// TwinCAT 3 PLC project PLC1
// Title: XPlanar Example Project
// Company: Beckhoff Automation LLC
// ProjectVersion: 1.0.0
// ProgramVersion: 3.1.4023.0
// libraries:
//   SPT Base Types, * (Beckhoff Automation LLC)
//   SPT Event Logger, * (Beckhoff Automation LLC)
//   SPT_XPlanar, * (Beckhoff Automation LLC)
//   Tc2_EtherCAT, * (Beckhoff Automation GmbH)
//   Tc2_Math, * (Beckhoff Automation GmbH)
//   Tc2_Standard, * (Beckhoff Automation GmbH)
//   Tc2_System, * (Beckhoff Automation GmbH)
//   Tc3_EventLogger, * (Beckhoff Automation GmbH)
//   Tc3_Module, * (Beckhoff Automation GmbH)
//   Tc3_PackML_V2, * (Beckhoff Automation GmbH)
//   Tc3_XPlanarUtility, * (Beckhoff Automation GmbH & Co. KG)
//   Tc3_Mc3PlanarMotion,newest,Beckhoff Automation GmbH
//   Tc3_Physics,newest,Beckhoff Automation GmbH
//   Tc3_XPlanarStandard,newest,Beckhoff Automation GmbH
//   VisuSymbols,3.5.10.0,System
// project tree:
//   / GlobalTextList.TcGTLO, MAIN.TcPOU, NextMinorStep.TcPOU, NextStep.TcPOU, PlcTask.TcTTO, StationList_TextList.TcTLO, Visualization Manager.TcVMO (not stored)
//   Machine/EquipmentModules/CustomStations/ FB_DecisionStation.TcPOU, FB_SpinStation.TcPOU
//   Machine/EquipmentModules/ FB_XPlanar_EM.TcPOU
//   Machine/ FB_Machine.TcPOU
//   Machine/VISUs/VisuOjects/ V_MachineModule.TcVIS, V_Module.TcVIS, V_Mover.TcVIS, V_RotaryAxis.TcVIS, V_Station.TcVIS
//   Machine/VISUs/ V_Main.TcVIS
// real-time tasks:
//   TASK PlcTask: cycle T#10ms, priority 20, ADS port 350
//   TASK Job Task: cycle default, priority 15
//   TASK MC-Task (MET): cycle T#2ms, priority 13, ADS port 521
//   TASK MC-Task (MPT): cycle T#10ms, priority 14, ADS port 531
//   TASK XPlanar Task11: cycle T#500us, priority 2, ADS port 352
//   TASK XPlanar Task6: cycle T#250us, priority 1, ADS port 351
//   TASK XPlanar Task7: cycle T#250us, priority 12, ADS port 353
//   TASK XPlanar Task3: cycle T#250us, priority 5, ADS port 354
//   TASK XPlanar Task4: cycle T#250us, priority 9, ADS port 355
//   TASK XPlanar Task5: cycle T#250us, priority 10, ADS port 356
// variable links:
//   XPlanar MC Project/Axes/Mover4220_1 <-> TcCOM Objects/XPlanar/Mover4220_1
//     McToIo/STD <-> InputsFromNC3/NC3ToHW
//   XPlanar MC Project/Axes/Mover4220_2 <-> TcCOM Objects/XPlanar/Mover4220_2
//     IoToMc/STD <-> OutputsToNC3/HWToNC3
//   XPlanar MC Project/Axes/Mover4220_3 <-> TcCOM Objects/XPlanar/Mover4220_3
//     IoToMc/STD <-> OutputsToNC3/HWToNC3
//   XPlanar MC Project/Axes/Mover4220_4 <-> TcCOM Objects/XPlanar/Mover4220_4
//     IoToMc/STD <-> OutputsToNC3/HWToNC3
//   PLC1/PLC1 Instance <-> XPlanar MC Project/Axes/Mover4220_1
//     PlcTask Inputs/MAIN.Machine.XPlanar.Movers[1]._Mover.stMoverRef.MCTOPLC/ACT <-> McToPlc/ACT
//     PlcTask Inputs/MAIN.Machine.XPlanar.Movers[1]._Mover.stMoverRef.MCTOPLC/COORDMODE <-> McToPlc/COORDMODE
//     PlcTask Inputs/MAIN.Machine.XPlanar.Movers[1]._Mover.stMoverRef.MCTOPLC/SET <-> McToPlc/SET
//     PlcTask Inputs/MAIN.Machine.XPlanar.Movers[1]._Mover.stMoverRef.MCTOPLC/SETONTRACK <-> McToPlc/SETONTRACK
//     PlcTask Inputs/MAIN.Machine.XPlanar.Movers[1]._Mover.stMoverRef.MCTOPLC/STD <-> McToPlc/STD
//     PlcTask Outputs/MAIN.Machine.XPlanar.Movers[1]._Mover.stMoverRef.PLCTOMC/STD <-> PlcToMc/STD
//   PLC1/PLC1 Instance <-> XPlanar MC Project/Axes/Mover4220_2
//     PlcTask Inputs/MAIN.Machine.XPlanar.Movers[2]._Mover.stMoverRef.MCTOPLC/ACT <-> McToPlc/ACT
//     PlcTask Inputs/MAIN.Machine.XPlanar.Movers[2]._Mover.stMoverRef.MCTOPLC/COORDMODE <-> McToPlc/COORDMODE
//     PlcTask Inputs/MAIN.Machine.XPlanar.Movers[2]._Mover.stMoverRef.MCTOPLC/SET <-> McToPlc/SET
//     PlcTask Inputs/MAIN.Machine.XPlanar.Movers[2]._Mover.stMoverRef.MCTOPLC/SETONTRACK <-> McToPlc/SETONTRACK
//     PlcTask Inputs/MAIN.Machine.XPlanar.Movers[2]._Mover.stMoverRef.MCTOPLC/STD <-> McToPlc/STD
//     PlcTask Outputs/MAIN.Machine.XPlanar.Movers[2]._Mover.stMoverRef.PLCTOMC/STD <-> PlcToMc/STD
//   PLC1/PLC1 Instance <-> XPlanar MC Project/Axes/Mover4220_3
//     PlcTask Inputs/MAIN.Machine.XPlanar.Movers[3]._Mover.stMoverRef.MCTOPLC/ACT <-> McToPlc/ACT
//     PlcTask Inputs/MAIN.Machine.XPlanar.Movers[3]._Mover.stMoverRef.MCTOPLC/COORDMODE <-> McToPlc/COORDMODE
//     PlcTask Inputs/MAIN.Machine.XPlanar.Movers[3]._Mover.stMoverRef.MCTOPLC/SET <-> McToPlc/SET
//     PlcTask Inputs/MAIN.Machine.XPlanar.Movers[3]._Mover.stMoverRef.MCTOPLC/SETONTRACK <-> McToPlc/SETONTRACK
//     PlcTask Inputs/MAIN.Machine.XPlanar.Movers[3]._Mover.stMoverRef.MCTOPLC/STD <-> McToPlc/STD
//     PlcTask Outputs/MAIN.Machine.XPlanar.Movers[3]._Mover.stMoverRef.PLCTOMC/STD <-> PlcToMc/STD
//   PLC1/PLC1 Instance <-> XPlanar MC Project/Axes/Mover4220_4
//     PlcTask Inputs/MAIN.Machine.XPlanar.Movers[4]._Mover.stMoverRef.MCTOPLC/ACT <-> McToPlc/ACT
//     PlcTask Inputs/MAIN.Machine.XPlanar.Movers[4]._Mover.stMoverRef.MCTOPLC/COORDMODE <-> McToPlc/COORDMODE
//     PlcTask Inputs/MAIN.Machine.XPlanar.Movers[4]._Mover.stMoverRef.MCTOPLC/SET <-> McToPlc/SET
//     PlcTask Inputs/MAIN.Machine.XPlanar.Movers[4]._Mover.stMoverRef.MCTOPLC/SETONTRACK <-> McToPlc/SETONTRACK
//     PlcTask Inputs/MAIN.Machine.XPlanar.Movers[4]._Mover.stMoverRef.MCTOPLC/STD <-> McToPlc/STD
//     PlcTask Outputs/MAIN.Machine.XPlanar.Movers[4]._Mover.stMoverRef.PLCTOMC/STD <-> PlcToMc/STD
//   PLC1/PLC1 Instance <-> XPlanar MC Project/Groups/Environment
//     PlcTask Inputs/MAIN.Machine.XPlanar.XPlanarTable.XPlanarSystem.environment.MCTOPLC_STD <-> McToPlc/STD
//   PLC1/PLC1 Instance <-> XPlanar MC Project/Groups/Group3 (Planar Track)
//     PlcTask Inputs/MAIN.Machine.XPlanar.Tracks[1].TrackStandard.stTrackRef.MCTOPLC_STD <-> McToPlc/STD
//   PLC1/PLC1 Instance <-> XPlanar MC Project/Groups/Group4 (Planar Track)
//     PlcTask Inputs/MAIN.Machine.XPlanar.Tracks[2].TrackStandard.stTrackRef.MCTOPLC_STD <-> McToPlc/STD
//   PLC1/PLC1 Instance <-> XPlanar MC Project/Groups/Group5 (Planar Track)
//     PlcTask Inputs/MAIN.Machine.XPlanar.Tracks[3].TrackStandard.stTrackRef.MCTOPLC_STD <-> McToPlc/STD
//   PLC1/PLC1 Instance <-> XPlanar MC Project/Groups/Group6 (Planar Track)
//     PlcTask Inputs/MAIN.Machine.XPlanar.Tracks[4].TrackStandard.stTrackRef.MCTOPLC_STD <-> McToPlc/STD
//   PLC1/PLC1 Instance <-> XPlanar MC Project/Groups/XPlanar
//     PlcTask Inputs/MAIN.Machine.XPlanar.XPlanarTable.XPlanarSystem.group.MCTOPLC_STD <-> McToPlc/STD
//   TcCOM Objects/XPlanar/Mover4220_1 <-> XPlanar MC Project/Axes/Mover4220_1
//     OutputsToNC3/HWToNC3 <-> IoToMc/STD
//   TcCOM Objects/XPlanar/Mover4220_2 <-> XPlanar MC Project/Axes/Mover4220_2
//     InputsFromNC3/NC3ToHW <-> McToIo/STD
//   TcCOM Objects/XPlanar/Mover4220_3 <-> XPlanar MC Project/Axes/Mover4220_3
//     InputsFromNC3/NC3ToHW <-> McToIo/STD
//   TcCOM Objects/XPlanar/Mover4220_4 <-> XPlanar MC Project/Axes/Mover4220_4
//     InputsFromNC3/NC3ToHW <-> McToIo/STD

CONFIGURATION PLC1
    RESOURCE PLC ON TwinCAT3
        TASK PlcTask(INTERVAL := T#10ms, PRIORITY := 20);
        PROGRAM MAIN WITH PlcTask : MAIN;
    END_RESOURCE
END_CONFIGURATION

// ---- MAIN.TcPOU

PROGRAM MAIN
VAR
    // Machine Module
    Machine : FB_Machine := (Name := 'My First XPlanar Component Project');
    //Control Source for running machine
    ControlSourceHMI : FB_ControlSource;
    ControlSourcePB  : FB_ControlSource;
    //Local Vars
    InitComplete : BOOL;
END_VAR

{warning 'Simulation Demo Only - Lag monitoring is disabled'}

//All code runs from here.
CyclicLogic();

METHOD CyclicLogic
VAR_INPUT
END_VAR
IF NOT InitComplete THEN
    InitComplete := Initialize();
    RETURN;
END_IF

//Machine support HMI & Production Monitor
ControlSourcePB.CyclicLogic();
ControlSourceHMI.CyclicLogic();

//Machine Cyclic Logic
Machine.CyclicLogic();
END_METHOD

METHOD Initialize : BOOL
VAR_INPUT
END_VAR

VAR
    Result : BOOL;
END_VAR
//Top level machine initialization should happen here, in the main initialization METHOD. Each subsequent "layer" OF modules will be named within their respective "parent" intialize METHOD
IF NOT ControlSourceHMI.Registered THEN
    Result := Machine.RegisterExternalController(ControlSourceHMI);
END_IF

IF NOT ControlSourcePB.Registered THEN
    Result := Machine.RegisterExternalController(ControlSourcePB);
END_IF

ControlSourceHMI.CyclicLogic();
ControlSourcePB.CyclicLogic();

ADSLOGSTR(ADSLOG_MSGTYPE_WARN, 'Lag Monitoring disabled', 'For simulation demo only',);

Initialize := TRUE;
END_METHOD

END_PROGRAM

// ---- Machine/FB_Machine.TcPOU
FUNCTION_BLOCK FB_Machine EXTENDS FB_PackML_BaseModule
VAR
    (*Sub Modules*)
    XPlanar : FB_XPlanar_EM := (Name := 'XPlaner EM');

    (*Initial List of SubModules*)

    //Add list of EMs here...
    ipSubModules_Init : ARRAY[1..Parameters_PackML_Base.MAX_NO_OF_SUBMODULES] OF I_PackML_BaseModule := [XPlanar];

    // Components

    //Add list of components here...
    ipComponents_Init : ARRAY[1..Parameters_PackML_Base.MAX_NO_OF_COMPONENTS] OF I_ComponentBase := [];

    // Local and Simulation variables

    (*Alarms for this module*)
    MachineAlarms : ARRAY[1..MACHINE_ALARM_COUNT] OF FB_TcAlarm;
    RecipeLoaded  : BOOL := FALSE;

    //Pack Tags for System
    {attribute 'OPC.UA.DA' := '1'}
    _PackTags : ST_PackMLv30Ext; //ST_PackMLv30 is obsolete in Tc3_PackML_V2
END_VAR

VAR CONSTANT
    //Alarm count constant
    MACHINE_ALARM_COUNT : INT := 1; //Change this value based on how many alarms are in your machine
END_VAR

METHOD PROTECTED CreateEvents
VAR_INPUT
END_VAR
// Add your event creation here
F_CreateAllEventsInClass(Alarms     := MachineAlarms,
                         ClassSize  := SIZEOF(TC_EVENTS.MachineAlarms),
                         pInitEvent := ADR(TC_EVENTS.MachineAlarms.InitReferenceEvent),
                         Prefix     := Name);

// Super call to base
SUPER^.CreateEvents();
END_METHOD

METHOD CyclicLogic
VAR
    NewSeverity    : TCEventSeverity;
    AlarmResponses : ARRAY[0..4] OF E_AlarmResponse; //Temporary response array	
END_VAR
IF NOT _InitComplete THEN
    _InitComplete := Initialize();
    RETURN;
END_IF

_CurrentAlarmSeverity := F_GetMaxSeverityRaised(MachineAlarms, NewSeverity);
SUPER^.CyclicLogic();
_PackTags.Status.StateCurrent    := _CurrentState;
_PackTags.Status.UnitModeCurrent := _CurrentMode;
UpdateModeTimers();
END_METHOD

METHOD PROTECTED HMIPermissions
VAR_INPUT
END_VAR
//General Mode Based Monitoring and handling of HMI control
CASE _CurrentMode OF
    E_PMLUnitMode.ePMLUnitMode_Production:
        CASE _CurrentState OF
            E_PMLState.ePMLState_Stopped:
                AllowHMIControl(ThisModuleOnly := TRUE); //Allow control for recovery
            E_PMLState.ePMLState_Idle:
                AllowHMIControl(ThisModuleOnly := TRUE); //Allow control for recovery
            E_PMLState.ePMLState_Suspended:
                BlockHMIControl();

            E_PMLState.ePMLState_Execute:
                BlockHMIControl();

            E_PMLState.ePMLState_Aborted:
                AllowHMIControl(ThisModuleOnly := TRUE); //Allow control for recovery
            E_PMLState.ePMLState_Held:
                AllowHMIControl(ThisModuleOnly := TRUE); //Allow control for recovery
            E_PMLState.ePMLState_Complete:
                BlockHMIControl();
        END_CASE

        AllowHMIControl(ThisModuleOnly := FALSE);

    E_PMLUnitMode.ePMLUnitMode_Manual:
        AllowHMIControl(ThisModuleOnly := FALSE);

    E_PMLUnitMode.ePMLUnitMode_Maintenance:
        AllowHMIControl(ThisModuleOnly := FALSE);
END_CASE
END_METHOD

METHOD PROTECTED Initialize : BOOL
VAR
    i : UDINT; //Generic iteration value
END_VAR
Initialize := FALSE;
CASE DescendantSequenceState OF
    0:
        // Define the interfaces to the different subunits (Must take place before SUPER^.initialize call)
        FOR i := 1 TO SPT_BaseTypes.Parameters_PackML_Base.MAX_NO_OF_SUBMODULES DO
            ipSubModules[i] := ipSubModules_Init[i];
        END_FOR

        FOR i := 1 TO SPT_BaseTypes.Parameters_PackML_Base.MAX_NO_OF_COMPONENTS DO
            ipComponents[i] := ipComponents_Init[i];
        END_FOR

        _LogModeChanges         := FALSE;
        _LogStateChanges        := FALSE;
        DescendantSequenceState := DescendantSequenceState + 10;

    10:
        //Setup Custom modes here
        DescendantSequenceState := DescendantSequenceState + 10;

    20:
        //Copy Mode names
        FOR i := 1 TO 3 DO
            ModeNames[i] := F_UnitModeToString(UDINT_TO_DINT(i));
        END_FOR

        DescendantSequenceState := DescendantSequenceState + 10;

    30:
        // Initialize Recipes 
        DescendantSequenceState := DescendantSequenceState + 10;

    40:
        //Call the Super
        IF SUPER^.Initialize() THEN
            DescendantSequenceState := DescendantSequenceState + 10;
        END_IF

    //Setup axes Master
    50:
        Initialize := TRUE;
END_CASE
END_METHOD

PROPERTY PUBLIC PackTags : ST_PackMLv30Ext
GET
PackTags := _PackTags;
END_GET
END_PROPERTY

//! @summary Provides fault reaction logic where the module state is driven to the <b>Stopping</b> state immediately
METHOD PROTECTED StopImmediate

//! @description No error is thrown by this fault reaction.

//! @description This method is called by <c>ComponentMonitor()</c> or <c>SubModuleMonitor()</c> as required
ChangeState(E_PMLCommand.ePMLCommand_Stop);
END_METHOD

METHOD PROTECTED SubModuleMonitor : BOOL
VAR
    AlarmResponses : ARRAY[0..4] OF E_AlarmResponse; //Temporary response array	
END_VAR

VAR
    Result : BOOL;
END_VAR
SubModuleMonitor := FALSE;

// Check the sub Modules for Alarm Severity
Result := SUPER^.SubModuleMonitor();

//Check the alarms at the machine level
_CurrentAlarmSeverity := F_GetMaxSeverityRaised(Alarms := MachineAlarms, CurrentSeverity := _CurrentAlarmSeverity);

//Check the severity of the machine level alarms
IF _CurrentState <> E_PMLState.ePMLState_Aborted AND _CurrentState <> E_PMLState.ePMLState_Aborting AND _CurrentState <> E_PMLState.ePMLState_Clearing AND
   _CurrentState <> E_PMLState.ePMLState_Stopped AND _CurrentState <> E_PMLState.ePMLState_Stopping THEN
    AlarmResponses := _ParentFaultResponseDefinitions;
    CASE AlarmResponses[CurrentAlarmSeverity] OF
        E_AlarmResponse.Abort_ImmediateError:
            AbortImmediateError(Name, TRUE);

        E_AlarmResponse.Abort_Immediate:
            AbortImmediate();

        E_AlarmResponse.Stop_Immediate:
            StopImmediate();

        E_AlarmResponse.Stop_Controlled:
            StopControlled();

        E_AlarmResponse.Hold_Immediate:
            HoldImmediate();

        E_AlarmResponse.Suspend_Immediate:
            SuspendImmediate();

        E_AlarmResponse.Suspend_Controlled:
            SuspendControlled();

        E_AlarmResponse.NoResponse:
            ;
    END_CASE
ELSIF _CurrentState = E_PMLState.ePMLState_Stopped OR _CurrentState = E_PMLState.ePMLState_Stopping THEN
    AlarmResponses := _ParentFaultResponseDefinitions;
    CASE AlarmResponses[CurrentAlarmSeverity] OF
        E_AlarmResponse.Abort_ImmediateError:
            AbortImmediateError(Name, TRUE);

        E_AlarmResponse.Abort_Immediate:
            AbortImmediate();

        E_AlarmResponse.NoResponse:
            ;
    END_CASE
END_IF
END_METHOD

METHOD UpdateModeTimers
VAR
    currentTime  : T_DCTIME64;
    timeToUpdate : LREAL;
END_VAR

VAR_INST
    lastTime  : T_DCTIME64 := F_GetActualDcTime64();
    lastState : DINT;
    lastMode  : DINT;
END_VAR

VAR
    Result : UDINT;
END_VAR
IF _PackTags.Status.StateCurrent <> lastState THEN
    Result    := MEMSET(ADR(_PackTags.Admin.StateCurrentTime), 0, SIZEOF(_PackTags.Admin.StateCurrentTime));
    lastState := _PackTags.Status.StateCurrent;
END_IF

IF _PackTags.Status.UnitModeCurrent <> lastMode THEN
    Result   := MEMSET(ADR(_PackTags.Admin.ModeCurrentTime), 0, SIZEOF(_PackTags.Admin.ModeCurrentTime));
    lastMode := _PackTags.Status.UnitModeCurrent;
END_IF

currentTime := F_GetActualDcTime64();
IF lastTime <> 0 THEN
    timeToUpdate := ULINT_TO_LREAL(currentTime - lastTime) / 1_000_000_000.0;
END_IF

// only seconds get added to the cumulative timers 
IF timeToUpdate > 1 THEN
    _PackTags.Admin.ModeCummulativeTime[_PackTags.Status.UnitModeCurrent] := _PackTags.Admin.ModeCummulativeTime[_PackTags.Status.UnitModeCurrent] + LREAL_TO_DINT(timeToUpdate);
    _PackTags.Admin.ModeCurrentTime[_PackTags.Status.UnitModeCurrent]     := _PackTags.Admin.ModeCurrentTime[_PackTags.Status.UnitModeCurrent] + LREAL_TO_DINT(timeToUpdate);
    _PackTags.Admin.StateCummulativeTime[_PackTags.Status.UnitModeCurrent, _PackTags.Status.StateCurrent]
        := _PackTags.Admin.StateCummulativeTime[_PackTags.Status.UnitModeCurrent, _PackTags.Status.StateCurrent] + LREAL_TO_DINT(timeToUpdate);

    _PackTags.Admin.StateCurrentTime[_PackTags.Status.UnitModeCurrent, _PackTags.Status.StateCurrent] :=
        _PackTags.Admin.StateCurrentTime[_PackTags.Status.UnitModeCurrent, _PackTags.Status.StateCurrent] + LREAL_TO_DINT(timeToUpdate);

    lastTime := currentTime;
END_IF
END_METHOD

END_FUNCTION_BLOCK

// ---- Machine/EquipmentModules/FB_XPlanar_EM.TcPOU
FUNCTION_BLOCK FB_XPlanar_EM EXTENDS FB_PackML_BaseModule
VAR
    // Sub module definitions here

    // List of sub modules
    ipSubModules_Init : ARRAY[1..Parameters_PackML_Base.MAX_NO_OF_SUBMODULES] OF I_PackML_BaseModule := [];

    // Component definitions here
    XPlanarTable : FB_Component_Xplanar := (Name := 'XPlanarTable');
	
	//Station Components
	Station1	 : FB_DecisionStation	 := (Name := 'DecisionPoint');   //Declaration of a custom station
	Station2	 : FB_SpinStation 		 := (Name := 'RotateStation');
	Station3	 : FB_XPlanarStationBase := (Name := 'InspectStation');  //If no custom processing is needed simply declare an instance of the Station Base fb	 

    // List of Components
    ipComponents_Init : ARRAY[1..Parameters_PackML_Base.MAX_NO_OF_COMPONENTS] OF I_ComponentBase := [XPlanarTable, Station1, Station2, Station3];

    //Helper Vars
	Movers			  : ARRAY[1..Tc3_XPlanarStandard.Params_XPlanar.moverCount] OF FB_XPlanarMover;
	Tracks			  : ARRAY[1..Tc3_XPlanarStandard.Params_XPlanar.maxTrackCount] OF FB_XPlanarTrackSegment;
END_VAR

//! @summary This method contains code which will execute when this PackML module is in the <b>Aborting</b> state
METHOD PROTECTED Aborting
VAR
    i               : UDINT;
    SubModulesReady : BOOL := TRUE;
END_VAR

(*! <description> <b>Note:</b> The <i>Abort</i> command should be associated with the fault handing routine of a module. It should not be directly commanded from any user inteface. 

<table> 
	<tr>
		<th> Previous State </th>
		<th> Transition In </th>
		<th> Transition Out </th>
		<th> Next State  </th> 
	</tr>
	<tr>
		<td> <b>ANY</b> </td>
		<td> Abort Command </td> 
		<td> State Complete </td>
		<td> Aborted </td> 
	</tr>
</table>

This method is called as required by <c>StateControl()</c>
</description> 

*)
CASE DescendantSequenceState OF
    0:
        NoStateTasksToComplete  := FALSE;
        DescendantSequenceState := NextStep(DescendantSequenceState);

    10:
        IF XPlanarTable.Abort() THEN
            StateTasksComplete      := TRUE;
            DescendantSequenceState := NextStep(DescendantSequenceState);
        END_IF

    20:
        StateTasksComplete := TRUE;
END_CASE

SUPER^.Aborting();
END_METHOD

//! @summary This method contains code which will execute when this PackML module is in the <b>Clearing</b> state
METHOD PROTECTED Clearing
VAR
    i               : UDINT;
    SubModulesReady : BOOL := TRUE;
END_VAR

(*! <description> <b>Note:</b> The <i>Clear</i> command can also be thought of as a <i>fault reset</i> depite the ambiguity in the naming of the <i>Reset</i> state. 
<table> 
	<tr>
		<th> Previous State </th>
		<th> Transition In </th>
		<th> Transition Out </th>
		<th> Next State  </th> 
	</tr>
	<tr>
		<td> Aborted </td>
		<td> Clear Command </td> 
		<td> State Complete </td>
		<td> Stopped </td> 
	</tr>
</table>
This method is called as required by <c>StateControl()</c>
</description> 

*)
CASE _CurrentMode OF
    E_PMLUnitMode.ePMLUnitMode_Production:
        CASE DescendantSequenceState OF
            0: //Init
                NoStateTasksToComplete  := FALSE;
                XPlanarTable._Error     := FALSE;
				Station1.Reset();
				Station2.Reset();
				Station3.Reset();
			
                DescendantSequenceState := NextStep(DescendantSequenceState);

            10: //Check for Track initialization
                IF NOT XPlanarTable.TracksInitialized THEN
                    DescendantSequenceState := NextMinorStep(DescendantSequenceState);
                ELSE
                    DescendantSequenceState := NextStep(DescendantSequenceState);
                END_IF

            11: //Build Track Segments
                IF XPlanarTable.BuildTracks() THEN
                    IF NOT XPlanarTable.Error THEN
                      DescendantSequenceState := NextStep(DescendantSequenceState);
                    ELSE
                        DescendantSequenceState := 999;
                    END_IF;
                END_IF

            20: //Enable Group
                IF XPlanarTable.EnableGroup() THEN
                    DescendantSequenceState := NextStep(DescendantSequenceState);
                END_IF

            30:
                //Clearing complete
                StateTasksComplete := TRUE;
        END_CASE

    E_PMLUnitMode.ePMLUnitMode_Manual:
        ;
END_CASE

SUPER^.Clearing();
END_METHOD

METHOD PROTECTED CreateEvents
VAR_INPUT
END_VAR
// Add your event creation here

// Super call to base
SUPER^.CreateEvents();
END_METHOD

METHOD CyclicLogic
VAR
    i : INT;
    j : UDINT;
END_VAR
IF NOT _InitComplete THEN
    _InitComplete := Initialize();
END_IF

SUPER^.CyclicLogic();
END_METHOD

//! @summary This method contains code which will execute when this PackML module is in the <b>Execute</b> state
METHOD PROTECTED Execute
VAR
    i : UDINT;
END_VAR
VAR_INST
	InspectSimTimer: TON;
END_VAR
(*! <description> <b>The base implementation of this method is empty. User must override this method to provide functionality.</b>
<table> 
	<tr>
		<th> Previous State </th>
		<th> Transition In </th>
		<th> Transition Out </th>
		<th> Next State  </th> 
	</tr>
	<tr>
		<td> Starting<b>-or-</b>Unholding <b>-or-</b>Unsuspending</td>
		<td> State Complete<i>(Starting<b>-or-</b>Unholding<b>-or-</b>Unsuspending)</i></td> 
		<td> State Complete<b>-or-</b>Hold Command<b>-or-</b>Suspend Command</td>
		<td> Completing<b>-or-</b>Holding<b>-or-</b>Suspending</td>
	</tr>
</table>
This method is called as required by <c>StateControl()</c>
</description> 

*)
CASE _CurrentMode OF
    E_PMLUnitMode.ePMLUnitMode_Production:
        FOR i := 1 TO Params_XPlanar.maxNumStation DO
            ip.Stations[i].Execute();
        END_FOR
	
	//Simulate the "Inspection Done" signal
	InspectSimTimer(IN := ip.Stations[3].StationReady, PT := T#1S);
	ip.Stations[3].StationComplete := InspectSimTimer.Q;
	
    E_PMLUnitMode.ePMLUnitMode_Manual:
        ;
END_CASE
END_METHOD

//! @summary Automatically enables and disables HMI control based on the PackML mode
METHOD PROTECTED HMIPermissions

//! @description This method is called cyclically by <c>CyclicLogic()</c>
//General Mode Based Monitoring and handling of HMI control
CASE _CurrentMode OF
    E_PMLUnitMode.ePMLUnitMode_Production:
        AllowHMIControl(ThisModuleOnly := FALSE);

    E_PMLUnitMode.ePMLUnitMode_Manual:
        AllowHMIControl(ThisModuleOnly := FALSE);

    E_PMLUnitMode.ePMLUnitMode_Maintenance:
        AllowHMIControl(ThisModuleOnly := FALSE);
END_CASE
END_METHOD

//! @summary Basic module initialization logic
METHOD PROTECTED Initialize : BOOL;
VAR
    i                        : UDINT;
    varInfo                  : __SYSTEM.VAR_INFO;
    AllSubUnitsInitialized   : BOOL := TRUE;
    AllComponentsInitialized : BOOL := TRUE;
    tmpMoveDynamics          : ST_MoveDynamics;
    stHaltDynamics           : ST_HaltDynamics;
END_VAR

//! @description This method is called by <c>CyclicLogic()</c> as required
Initialize := FALSE;
CASE DescendantSequenceState OF
	0:
		// Define the interfaces to the different subunits (Must take place before SUPER^.initialize call)
		FOR i := 1 TO SPT_BaseTypes.Parameters_PackML_Base.MAX_NO_OF_SUBMODULES DO
			ipSubModules[i] := ipSubModules_Init[i];
		END_FOR

		FOR i := 1 TO SPT_BaseTypes.Parameters_PackML_Base.MAX_NO_OF_COMPONENTS DO
			ipComponents[i] := ipComponents_Init[i];
		END_FOR

		_LogModeChanges			:= FALSE;
		_LogStateChanges		:= FALSE;
		DescendantSequenceState := DescendantSequenceState + 10;

	10:
		//Set Mover and Track interfaces
		FOR i := 1 TO Tc3_XPlanarStandard.Params_XPlanar.moverCount DO
			Movers[i].MoverIndex := i;
			ip.Movers[i]		  := Movers[i];
		END_FOR

		FOR i := 1 TO Tc3_XPlanarStandard.Params_XPlanar.maxTrackCount DO
			ip.Tracks[i] := Tracks[i];
		END_FOR

		DescendantSequenceState := DescendantSequenceState + 10;

	20:
		//Copy Mode names
		FOR i := 1 TO 3 DO
			ModeNames[i] := F_UnitModeToString(UDINT_TO_DINT(i));
		END_FOR

		DescendantSequenceState := DescendantSequenceState + 10;

	30:
		//Call the Super
		IF SUPER^.Initialize() THEN
			DescendantSequenceState := DescendantSequenceState + 10;
		END_IF

	40:
		IF SetupTrackSegments() THEN
			DescendantSequenceState := DescendantSequenceState + 10;
		END_IF

	50:
		IF SetupStations() THEN
			DescendantSequenceState := DescendantSequenceState + 10;
		END_IF

	60:
		stHaltDynamics.PathXY.fVelocity		:= 500.0;
		stHaltDynamics.PathXY.fAcceleration := 10000.0;
		stHaltDynamics.PathXY.fDeceleration := 10000.0;
		stHaltDynamics.PathXY.fJerk			:= 100000.0;
		stHaltDynamics.AxisX.fVelocity		:= 500.0;
		stHaltDynamics.AxisX.fAcceleration	:= 10000.0;
		stHaltDynamics.AxisX.fDeceleration	:= 10000.0;
		stHaltDynamics.AxisX.fJerk			:= 100000.0;
		stHaltDynamics.AxisY.fVelocity		:= 500.0;
		stHaltDynamics.AxisY.fAcceleration	:= 10000.0;
		stHaltDynamics.AxisY.fDeceleration	:= 10000.0;
		stHaltDynamics.AxisY.fJerk			:= 100000.0;
		stHaltDynamics.AxisZ.fVelocity		:= 500.0;
		stHaltDynamics.AxisZ.fAcceleration	:= 10000.0;
		stHaltDynamics.AxisZ.fDeceleration	:= 10000.0;
		stHaltDynamics.AxisZ.fJerk			:= 100000.0;
		stHaltDynamics.AxisA.fVelocity		:= 10.0;
		stHaltDynamics.AxisA.fAcceleration	:= 100.0;
		stHaltDynamics.AxisA.fDeceleration	:= 100.0;
		stHaltDynamics.AxisA.fJerk			:= 100.0;
		stHaltDynamics.AxisB.fVelocity		:= 10.0;
		stHaltDynamics.AxisB.fAcceleration	:= 100.0;
		stHaltDynamics.AxisB.fDeceleration	:= 100.0;
		stHaltDynamics.AxisB.fJerk			:= 100.0;
		stHaltDynamics.AxisC.fVelocity		:= 36.0;
		stHaltDynamics.AxisC.fAcceleration	:= 360.0;
		stHaltDynamics.AxisC.fDeceleration	:= 360.0;
		stHaltDynamics.AxisC.fJerk			:= 360.0;
		FOR i := 1 TO Params_XPlanar.moverCount DO
			ip.Movers[i].std.P_HaltDynamics := stHaltDynamics;
		END_FOR

		Initialize := TRUE;
END_CASE
END_METHOD

//! @summary This method contains code which will execute when this PackML module is in the <b>Resetting</b> state
METHOD PROTECTED Resetting
VAR
	SubModulesReady : BOOL := TRUE;
END_VAR

VAR_INST
	i : UDINT;
END_VAR

(*! <description> <b>Note:</b> The <i>Reset</i> command can also be thought of as an <i>enable</i> depite the ambiguity in the naming of the <i>Clearing</i> state.
<table> 
	<tr>
		<th> Previous State </th>
		<th> Transition In </th>
		<th> Transition Out </th>
		<th> Next State  </th> 
	</tr>
	<tr>
		<td> Stopped<b>-or-</b>Completed </td>
		<td> Reset Command </td> 
		<td> State Complete </td>
		<td> Idle </td> 
	</tr>
</table>
This method is called as required by <c>StateControl()</c>
</description> 

*)
CASE _CurrentMode OF
	E_PMLUnitMode.ePMLUnitMode_Production:
		CASE DescendantSequenceState OF
			0: //Init
				i						:= 1;
				NoStateTasksToComplete	:= FALSE;
				DescendantSequenceState := NextStep(DescendantSequenceState);

			10: //Reset XPlanar System
				IF XPlanarTable.Reset() THEN
					DescendantSequenceState := NextStep(DescendantSequenceState);
				END_IF

			20: //Enable Tracks
				IF XplanarTable.EnableTracks(FALSE) THEN
					DescendantSequenceState := NextStep(DescendantSequenceState);
				END_IF

			30: //Enable Movers
				IF XPlanarTable.EnableMovers(FALSE) THEN
					DescendantSequenceState := NextStep(DescendantSequenceState);
				END_IF

			40: //Check Mover Angle
				IF i <= Params_XPlanar.moverCount THEN
					IF ip.Movers[1].SquareUp() THEN
						DescendantSequenceState := NextMinorStep(DescendantSequenceState);
					END_IF
				ELSE
					DescendantSequenceState := NextStep(DescendantSequenceState);
				END_IF
				
			41: //CheckMoverCount
				IF i <= Params_XPlanar.moverCount THEN
					i := i + 1;
					DescendantSequenceState := 40;
				ELSE
					DescendantSequenceState := NextStep(DescendantSequenceState);
				END_IF				

			50: //Clearing complete
				StateTasksComplete := TRUE;
		END_CASE
END_CASE

SUPER^.Resetting();
END_METHOD

METHOD PRIVATE SetupStations : BOOL
VAR_INPUT
END_VAR
//Set Required Process Station Initialization Parameters
Station1.Position.SetValuesXYC(120, 360, 0);		 //Set the center of the station
Station1.TrackID	 := ip.Tracks[1];				 //Set the interface of the track segment the station resides on
Station1.StationType := E_StationType.DecisionPoint; //Change the type to Decision Point only if the station is acting as a divert and processing on the fly
Station1.OutputA	 := Station2;					 //Set any custom station parameters
Station1.OutputB	 := Station3;
ip.Stations[1]		 := Station1; 					 //Register the station with the interface array

Station2.Position.SetValuesXYC(600, 360, 0);
Station2.Size.x		 := 120;						 //Changes the station size in the X plane
Station2.Size.y		 := 120; 						 //Changes the station size in the Y plane
Station2.TrackID	 := ip.Tracks[2];
Station2.NextStation := Station1; 					 //Set the interface for the next station of the mover
ip.Stations[2]		 := Station2;

Station3.Position.SetValuesXYC(840.0, 360.0, 0);
Station3.Size.x		 := 120;
Station3.Size.y		 := 120;
Station3.TrackID	 := ip.Tracks[3];
Station3.NextStation := Station1;
ip.Stations[3]		 := Station3;
SetupStations		 := TRUE;
END_METHOD

METHOD PRIVATE SetupTrackSegments : BOOL
VAR_INST
    nSegmentIndex : UDINT;
END_VAR

VAR
    ResultAddPoint : INT;
END_VAR
SetupTrackSegments := FALSE;
CASE nSegmentIndex OF
	0: //Get ready
		nSegmentIndex := nSegmentIndex + 1;

	//********************************************************************************************************************************

	//Add states for each track segment in the system

	//********************************************************************************************************************************
	1:
		ip.Tracks[nSegmentIndex].ID := nSegmentIndex;
		IF ip.Tracks[nSegmentIndex].TrackTable.ClearTrackTable() THEN
			ResultAddPoint := ip.Tracks[nSegmentIndex].TrackTable.AddPoint(E_PointType.Line_Start,
																		   E_PointOption.none,
																		   480.0,
																		   120.0,
																		   0.0);

			ResultAddPoint := ip.Tracks[nSegmentIndex].TrackTable.AddPoint(E_PointType.Line_End,
																		   E_PointOption.none,
																		   240.0,
																		   120.0,
																		   0.0);

			ResultAddPoint := ip.Tracks[nSegmentIndex].TrackTable.AddPoint(E_PointType.Line_Start,
																		   E_PointOption.none,
																		   120.0,
																		   240.0,
																		   0.0);

			ResultAddPoint := ip.Tracks[nSegmentIndex].TrackTable.AddPoint(E_PointType.Line_End,
																		   E_PointOption.none,
																		   120.0,
																		   480.0,
																		   0.0);

			ResultAddPoint := ip.Tracks[nSegmentIndex].TrackTable.AddPoint(E_PointType.Line_Start,
																		   E_PointOption.none,
																		   240.0,
																		   600.0,
																		   0.0);

			ResultAddPoint := ip.Tracks[nSegmentIndex].TrackTable.AddPoint(E_PointType.Line_End,
																		   E_PointOption.none,
																		   480.0,
																		   600.0,
																		   0.0);

			ip.Tracks[nSegmentIndex].TrackTable.P_CloseTheLoop := FALSE;
		END_IF

		nSegmentIndex := nSegmentIndex + 1;

	2:
		ip.Tracks[2].ID := 2;  															//Set the ID property of the track segment
		IF ip.Tracks[2].TrackTable.ClearTrackTable() THEN								//Clean up any stray points in the table
			ResultAddPoint := ip.Tracks[2].TrackTable.AddPoint(E_PointType.Line_Start,	//Configure track points
															   E_PointOption.none,
															   600.0,
															   480.0,
															   0.0);

			ResultAddPoint := ip.Tracks[2].TrackTable.AddPoint(E_PointType.Line_End,
															   E_PointOption.none,
															   600.0,
															   240.0,
															   0.0);

			ip.Tracks[2].TrackTable.P_CloseTheLoop	 := FALSE;						//Set the segment close the loop property		
			ip.Tracks[2].TrackTable.P_StartFromTrack := ip.Tracks[1].std;			//If linking to a previous track segment set the interface
			ip.Tracks[2].TrackTable.P_EndAtTrack	 := ip.Tracks[1].std;			//If linking to a downstream track segment set the interface
		END_IF

		nSegmentIndex := nSegmentIndex + 1;

	3:
		ip.Tracks[nSegmentIndex].ID := nSegmentIndex;
		IF ip.Tracks[nSegmentIndex].TrackTable.ClearTrackTable() THEN
			ResultAddPoint := ip.Tracks[nSegmentIndex].TrackTable.AddPoint(E_PointType.Line_Start,
																		   E_PointOption.none,
																		   480.0,
																		   600.0,
																		   0.0);

			ResultAddPoint := ip.Tracks[nSegmentIndex].TrackTable.AddPoint(E_PointType.Line_End,
																		   E_PointOption.none,
																		   720.0,
																		   600.0,
																		   0.0);

			ResultAddPoint := ip.Tracks[nSegmentIndex].TrackTable.AddPoint(E_PointType.Line_Start,
																		   E_PointOption.none,
																		   840.0,
																		   480.0,
																		   0.0);

			ResultAddPoint := ip.Tracks[nSegmentIndex].TrackTable.AddPoint(E_PointType.Line_End,
																		   E_PointOption.none,
																		   840.0,
																		   240.0,
																		   0.0);

			ResultAddPoint := ip.Tracks[nSegmentIndex].TrackTable.AddPoint(E_PointType.Line_Start,
																		   E_PointOption.none,
																		   720.0,
																		   120.0,
																		   0.0);

			ResultAddPoint := ip.Tracks[nSegmentIndex].TrackTable.AddPoint(E_PointType.Line_End,
																		   E_PointOption.none,
																		   480.0,
																		   120.0,
																		   0.0);

			ip.Tracks[nSegmentIndex].TrackTable.P_CloseTheLoop	 := FALSE;
			ip.Tracks[nSegmentIndex].TrackTable.P_StartFromTrack := ip.Tracks[1].std;
			ip.Tracks[nSegmentIndex].TrackTable.P_EndAtTrack	 := ip.Tracks[1].std;
		END_IF

		nSegmentIndex := nSegmentIndex + 1;
		
	4:
		ip.Tracks[nSegmentIndex].ID := nSegmentIndex;
		IF ip.Tracks[nSegmentIndex].TrackTable.ClearTrackTable() THEN
			ResultAddPoint := ip.Tracks[nSegmentIndex].TrackTable.AddPoint(E_PointType.Line_Start,
																		   E_PointOption.none,
																		   100.0,
																		   100.0,
																		   0.0);

			ResultAddPoint := ip.Tracks[nSegmentIndex].TrackTable.AddPoint(E_PointType.Line_End,
																		   E_PointOption.none,
																		   100.0,
																		   500.0,
																		   0.0);

			ResultAddPoint := ip.Tracks[nSegmentIndex].TrackTable.AddPoint(E_PointType.Line_Start,
																		   E_PointOption.none,
																		   240.0,
																		   620.0,
																		   0.0);

			ResultAddPoint := ip.Tracks[nSegmentIndex].TrackTable.AddPoint(E_PointType.Line_End,
																		   E_PointOption.none,
																		   780.0,
																		   620.0,
																		   0.0);

			ResultAddPoint := ip.Tracks[nSegmentIndex].TrackTable.AddPoint(E_PointType.Line_Start,
																		   E_PointOption.none,
																		   860.0,
																		   480.0,
																		   0.0);

			ResultAddPoint := ip.Tracks[nSegmentIndex].TrackTable.AddPoint(E_PointType.Line_End,
																		   E_PointOption.none,
																		   860.0,
																		   240.0,
																		   0.0);
																		   
			ResultAddPoint := ip.Tracks[nSegmentIndex].TrackTable.AddPoint(E_PointType.Point,
																		   E_PointOption.none,
																		   860.0,
																		   240.0,
																		   0.0);																

			ip.Tracks[nSegmentIndex].TrackTable.P_CloseTheLoop	 := FALSE;
			ip.Tracks[nSegmentIndex].TrackTable.P_EndAtTrack	 := ip.Tracks[1].std;
		END_IF

		nSegmentIndex := nSegmentIndex + 1;		

	5:
		nSegmentIndex	   := 0;
		SetupTrackSegments := TRUE;
END_CASE
END_METHOD

//! @summary This method contains code which will execute when this PackML module is in the <b>Starting</b> state
METHOD PROTECTED Starting
VAR
    SubModulesReady : BOOL := TRUE;
    Position        : PositionXYC;
    check           : ST_CheckStartConditionFeedback;
    lError          : BOOL;
    lErrorID        : UDINT;
    Angle           : LREAL;
END_VAR

VAR_INST
    MoverNumber       : UDINT;
    StationNumber     : UDINT;
    ipMover           : I_XPlanarMover;
    ipStation         : I_XPlanarStation;
    JoinState         : INT;
    MoveState         : INT;
    i                 : UDINT;
    JoinTrackNum      : UINT;
    MoveStationNum    : ARRAY[1..Params_XPlanar.moverCount] OF UINT;
    MoveStationNeeded : ARRAY[1..Params_XPlanar.moverCount] OF BOOL;
    JoinStationNeeded : ARRAY[1..Params_XPlanar.moverCount] OF BOOL;
END_VAR
CASE _CurrentMode OF
	E_PMLUnitMode.ePMLUnitMode_Production:
		CASE DescendantSequenceState OF
			0:
				NoStateTasksToComplete	:= FALSE;
				DescendantSequenceState := 10;
				StationNumber			:= 1;
				i						:= 1;
				JoinState				:= 0;

			10: //Clean Up Mover Queues
				FOR i := 1 TO Params_XPlanar.moverCount DO
					ip.Movers[i].Destination := 0;
				END_FOR

				FOR i := 1 TO Params_XPlanar.maxNumStation DO
					ip.Stations[i].MoverQueue.Dequeue();
				END_FOR

				i						:= 1;
				DescendantSequenceState := NextStep(DescendantSequenceState);

			20: //Join Movers to recovery track
				IF i <= Params_XPlanar.moverCount THEN
					IF ip.Movers[i].JoinTrack(ip.Tracks[4]) THEN
						DescendantSequenceState := NextMinorStep(DescendantSequenceState);
					END_IF
				ELSE
					i						:= 1;
					DescendantSequenceState := NextStep(DescendantSequenceState);
				END_IF
				
			21: //Check Mover Count
				IF i <= Params_XPlanar.moverCount THEN
 					i := i + 1;
					DescendantSequenceState := 20;
				ELSE
					i						:= 1;
					DescendantSequenceState := NextStep(DescendantSequenceState);
				END_IF					

			30: //Send Movers around to station 1
				IF i <= Params_XPlanar.moverCount THEN
					IF ip.Movers[i].SendToStation(ip.Stations[1]) THEN
						DescendantSequenceState := NextMinorStep(DescendantSequenceState);
					END_IF
				ELSE
					i						:= 1;
					DescendantSequenceState := NextStep(DescendantSequenceState);
				END_IF
				
			31: //Check Mover Count
				IF i <= Params_XPlanar.moverCount THEN
 					i := i + 1;
					DescendantSequenceState := 30;
				ELSE
					i						:= 1;
					DescendantSequenceState := NextStep(DescendantSequenceState);
				END_IF	

			40:
				StateTasksComplete := TRUE;
		END_CASE

	E_PMLUnitMode.ePMLUnitMode_Manual:
		;
END_CASE

SUPER^.Starting();
END_METHOD

END_FUNCTION_BLOCK

// ---- Machine/EquipmentModules/CustomStations/FB_DecisionStation.TcPOU
FUNCTION_BLOCK FB_DecisionStation EXTENDS FB_XPlanarStationBase
VAR_INPUT
END_VAR
VAR_OUTPUT
END_VAR
VAR
	_OutputA	: I_XplanarStation;
	_OutputB	: I_XPlanarStation;
END_VAR

METHOD Execute
SUPER^.Execute(); //Call the base station logic to handle sending and receiving of movers

//When the station is in the Process mover state you can perform any application specific station logic
IF StationState = E_XPlanarStationState.ProcessMover THEN	
	IF ipCurrentMover.MoverIndex = 1 THEN			 
		ipNextStation := _OutputA;
	ELSE
		ipNextStation := _OutputB;
	END_IF
_StationComplete := TRUE;	//Set _StationComplete TRUE when done.  This will be automatically reset when the mover exits
END_IF
END_METHOD

PROPERTY OutputA : I_XPlanarStation
SET
_OutputA := OutputA;
END_SET
END_PROPERTY

PROPERTY OutputB : I_XPlanarStation
SET
_OutputB := OutputB;
END_SET
END_PROPERTY

END_FUNCTION_BLOCK

// ---- Machine/EquipmentModules/CustomStations/FB_SpinStation.TcPOU
FUNCTION_BLOCK FB_SpinStation EXTENDS FB_XPlanarStationBase
VAR_INPUT
END_VAR
VAR_OUTPUT
END_VAR
VAR
END_VAR

METHOD Execute
SUPER^.Execute();  //Call the base station logic to handle sending and receiving of movers

//When the station is in the Process mover state you can perform any application specific station logic
IF StationState = E_XPlanarStationState.ProcessMover THEN
	IF ipCurrentMover.Spin(NumOfTurns := 2) THEN
		_StationComplete := TRUE;  //Set _StationComplete TRUE when done.  This will be automatically reset when the mover exits
	END_IF
END_IF
END_METHOD

END_FUNCTION_BLOCK

// ---- NextStep.TcPOU
FUNCTION NextStep : UDINT
VAR_INPUT
	StateVar	: UDINT;
END_VAR
VAR
END_VAR

NextStep := ((StateVar / 10)* 10) + 10;

END_FUNCTION

// ---- NextMinorStep.TcPOU
FUNCTION NextMinorStep : UDINT
VAR_INPUT
	StateVar	: UDINT;
END_VAR
VAR
END_VAR

NextMinorStep := StateVar + 1;

END_FUNCTION

// ---- GlobalTextList.TcGTLO
TEXTLIST GlobalTextList
  996 = '%3.1f'
  188 = '%d'
  685 = '%s'
  309 = '%S'
  638 = '%x'
  508 = '%X'
  81 = '1'
  902 = '2'
  489 = '3'
  115 = '4'
  268 = '5'
  453 = 'A'
  680 = 'Abort'
  8 = 'B'
  122 = 'BAO Jam PE'
  139 = 'Bridge Breaker Down'
  111 = 'Bridge Breaker Up'
  557 = 'C'
  452 = 'Clear'
  276 = 'Disc Level PE'
  217 = 'Downstream Backup PE'
  280 = 'Enabled'
  54 = 'Exit Jam PE'
  316 = 'Fault'
  842 = 'Has Mover'
  944 = 'HMI PB Station'
  744 = 'Hold'
  53 = 'Home'
  551 = 'Hopper Level PE'
  182 = 'Initialized'
  938 = 'M1'
  303 = 'M2'
  38 = 'M3'
  609 = 'M4'
  347 = 'MACHINE'
  822 = 'MACHINE STATE CONTROL'
  46 = 'Maintenance'
  904 = 'Manual'
  114 = 'Mover'
  374 = 'Mover Fault'
  899 = 'Movers'
  463 = 'Number of Movers'
  78 = 'Number of Statinon'
  735 = 'Number of Statins'
  915 = 'Number of Stations'
  667 = 'Number of Tracks'
  49 = 'Operational Control Pad'
  880 = 'PowerOK'
  929 = 'Production'
  924 = 'Pushbutton Station'
  181 = 'Reset'
  252 = 'Send Away'
  780 = 'Speed Shift PE'
  77 = 'Start'
  839 = 'State-Machine Pad'
  516 = 'State: %s'
  739 = 'Stations'
  828 = 'Stop'
  806 = 'Suspend'
  386 = 'Tile Count'
  499 = 'Track'
  197 = 'Unhold'
  832 = 'Unsuspend'
  466 = 'Utility'
  785 = 'X'
  984 = 'XPlanar Example Project'
  88 = 'XPlanar Table'
  440 = 'Y'
  313 = 'y'
  438 = 'Z'
END_TEXTLIST

// ---- Machine/VISUs/VisuOjects/V_MachineModule.TcVIS
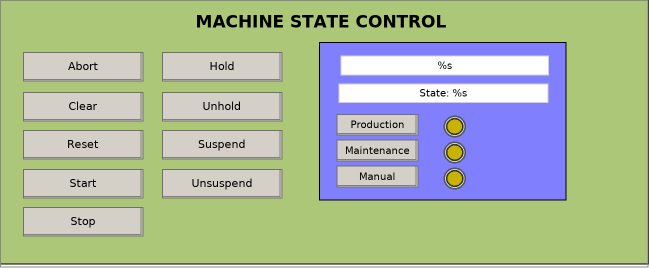
VISUALIZATION V_MachineModule  // 649x268
VAR_IN_OUT
	HMI : ST_PackMLBaseModule_HMI;
END_VAR
    RoundedRectangle (0,-4 649x268)
    Button (23,52 120x29), "Abort"
        OnMouseClick: execute { HMI.Command.State := E_PMLCommand.ePMLCommand_Abort; }
    Button (23,92 120x29), "Clear"
        OnMouseClick: execute { HMI.Command.State := E_PMLCommand.ePMLCommand_Clear; }
    Button (23,130 120x29), "Reset"
        OnMouseClick: execute { HMI.Command.State := E_PMLCommand.ePMLCommand_Reset; }
    Button (23,169 120x29), "Start"
        OnMouseClick: execute { HMI.Command.State := E_PMLCommand.ePMLCommand_Start; }
    Button (23,207 120x29), "Stop"
        OnMouseClick: execute { HMI.Command.State := E_PMLCommand.ePMLCommand_Stop; }
    Button (162,52 120x29), "Hold"
        OnMouseClick: execute { HMI.Command.State := E_PMLCommand.ePMLCommand_Hold; }
    Button (162,92 120x29), "Unhold"
        OnMouseClick: execute { HMI.Command.State := E_PMLCommand.ePMLCommand_Unhold; }
    Button (162,130 120x29), "Suspend"
        OnMouseClick: execute { HMI.Command.State := E_PMLCommand.ePMLCommand_Suspend; }
    Button (162,169 120x29), "Unsuspend"
        OnMouseClick: execute { HMI.Command.State := E_PMLCommand.ePMLCommand_Unsuspend; }
    Frame (319,42 247x158)
        shows V_Module(HMI := HMI)
    Label (31,3 580x37), "MACHINE STATE CONTROL"
END_VISUALIZATION

// ---- Machine/VISUs/VisuOjects/V_Module.TcVIS
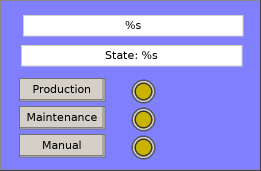
VISUALIZATION V_Module  // 261x171
VAR_IN_OUT
	HMI : ST_PackMLBaseModule_HMI;
END_VAR
    RoundedRectangle (0,0 261x171)
    Textfield (23,15 220x21), "%s", text variable: HMI.Config.Name
    Textfield (21,45 221x21), "State: %s", text variable: HMI.Status.State
    Button (19,78 86x23), "Production"
        OnMouseClick: execute { HMI.Command.Mode := E_PMLUnitMode.ePMLUnitMode_Production; }
    Button (19,106 86x23), "Maintenance"
        OnMouseClick: execute { HMI.Command.Mode := E_PMLUnitMode.ePMLUnitMode_Maintenance; }
    Button (19,134 86x23), "Manual"
        OnMouseClick: execute { HMI.Command.Mode := E_PMLUnitMode.ePMLUnitMode_Manual; }
    Lamp1 (130,78 27x27), variable: HMI.Status.Mode = E_PMLUnitMode.ePMLUnitMode_Production, style: Lamp-Lamp1-Yellow
    Lamp1 (130,106 27x27), variable: HMI.Status.Mode = E_PMLUnitMode.ePMLUnitMode_Maintenance, style: Lamp-Lamp1-Yellow
    Lamp1 (130,134 27x27), variable: HMI.Status.Mode = E_PMLUnitMode.ePMLUnitMode_Manual, style: Lamp-Lamp1-Yellow
END_VISUALIZATION

// ---- Machine/VISUs/VisuOjects/V_Mover.TcVIS
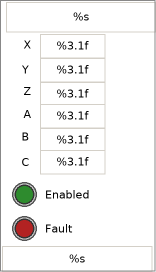
VISUALIZATION V_Mover  // 156x272
VAR_IN_OUT
	Mover : ST_Mover_HMI;
	Position : Position6D;
END_VAR
    Label (14,30 27x30), "X"
    Label (12,58 27x24), "Y"
    Label (14,80 27x23), "Z"
    Label (14,104 27x21), "A"
    Label (12,124 27x26), "B"
    Label (12,152 27x21), "C"
    Textfield (40,34 65x24), "%3.1f", text variable: Position.x
    Textfield (40,58 65x24), "%3.1f", text variable: Position.y
    Textfield (40,82 65x24), "%3.1f", text variable: Position.z
    Textfield (40,104 65x24), "%3.1f", text variable: Position.a
    Textfield (40,128 65x24), "%3.1f", text variable: Position.b
    Textfield (40,150 65x24), "%3.1f", text variable: Position.c
    Lamp1 (10,180 29x29), variable: Mover.Status.Enabled, style: Lamp-Lamp1-Green
    Label (42,182 107x26), "Enabled"
    Textfield (6,2 150x30), "%s", text variable: Mover.Status.ID
    Textfield (2,246 150x26), "%s", text variable: Mover.Status.CommandMode
    Lamp1 (10,214 29x29), variable: Mover.Status.Error, style: Lamp-Lamp1-Red
    Label (42,216 107x26), "Fault"
END_VISUALIZATION

// ---- Machine/VISUs/VisuOjects/V_RotaryAxis.TcVIS
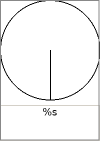
VISUALIZATION V_RotaryAxis  // 100x141
VAR_IN_OUT
	Axis : ST_AxisBase_HMI;
	Component : ST_ComponentBase_HMI;
END_VAR
    Ellipse (0,0 100x100)
    Line (50,50) (50,100)
        p2858320360: Axis.Status.ActualPositionModulo
    Textfield (0,105 100x36), "%s", text variable: Component.Config.Name
END_VISUALIZATION

// ---- Machine/VISUs/VisuOjects/V_Station.TcVIS
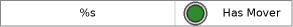
VISUALIZATION V_Station  // 293x27
VAR_IN_OUT
	Station : ST_Station_HMI;
END_VAR
    Textfield (0,0 175x26), "%s", text variable: Station.Status.MoverID
    Lamp1 (180,0 31x27), variable: Station.Status.HasMover, style: Lamp-Lamp1-Green
    Textfield (210,0 83x26), "Has Mover"
END_VISUALIZATION

// ---- Machine/VISUs/V_Main.TcVIS
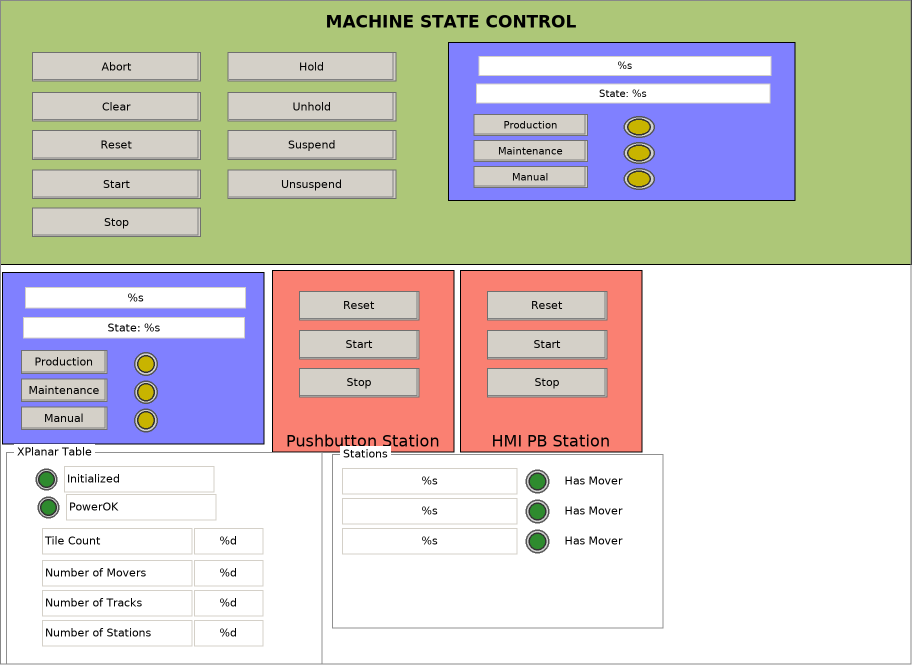
VISUALIZATION V_Main  // 912x665
    Frame (0,0 912x269)
        shows V_MachineModule(HMI := MAIN.Machine.PackMLBaseModule_HMI)
    Frame (2,272 262x172)
        shows V_Module(HMI := MAIN.Machine.XPlanar.PackMLBaseModule_HMI)
    Group (272,270 182x175)
        RoundedRectangle (0,0 182x182), "Pushbutton Station"
        Button (27,98 120x29), "Stop", input disabled if: not MAIN.ControlSourcePB.MainPMLControl_Simplified.StopPermissive
            tap MAIN.ControlSourcePB.MainPMLControl_Simplified.StopPressed
        Button (27,21 120x29), "Reset", input disabled if: not MAIN.ControlSourcePB.MainPMLControl_Simplified.ResetPermissive
            tap MAIN.ControlSourcePB.MainPMLControl_Simplified.ResetPressed
        Button (27,60 120x29), "Start", input disabled if: not MAIN.ControlSourcePB.MainPMLControl_Simplified.StartPermissive
            tap MAIN.ControlSourcePB.MainPMLControl_Simplified.StartPressed
    Group (460,270 182x175)
        RoundedRectangle (0,0 182x182), "HMI PB Station"
        Button (27,98 120x29), "Stop", input disabled if: not MAIN.ControlSourceHMI.MainPMLControl_Simplified.StopPermissive
            tap MAIN.ControlSourceHMI.MainPMLControl_Simplified.StopPressed
        Button (27,21 120x29), "Reset", input disabled if: not MAIN.ControlSourceHMI.MainPMLControl_Simplified.ResetPermissive
            tap MAIN.ControlSourceHMI.MainPMLControl_Simplified.ResetPressed
        Button (27,60 120x29), "Start", input disabled if: not MAIN.ControlSourceHMI.MainPMLControl_Simplified.StartPermissive
            tap MAIN.ControlSourceHMI.MainPMLControl_Simplified.StartPressed
    Group (332,446 331x219)
        Frame (10,22 293x27)
            shows V_Station(Station := MAIN.Machine.XPlanar.Station1.Station_HMI)
        Frame (10,52 293x27)
            shows V_Station(Station := MAIN.Machine.XPlanar.Station2.Station_HMI)
        Frame (10,82 293x27)
            shows V_Station(Station := MAIN.Machine.XPlanar.Station3.Station_HMI)
        GroupBox (0,0 331x182), "Stations"
    Group (6,444 316x220)
        Lamp1 (28,23 25x25), variable: MAIN.Machine.XPlanar.XPlanarTable.XPlanar_HMI.Status.Initialized, style: Lamp-Lamp1-Green
        Textfield (58,22 150x26), "Initialized"
        Lamp1 (30,51 25x25), variable: MAIN.Machine.XPlanar.XPlanarTable.XPlanar_HMI.Status.PowerOK, style: Lamp-Lamp1-Green
        Textfield (60,50 150x26), "PowerOK"
        Textfield (188,84 69x26), "%d", text variable: MAIN.Machine.XPlanar.XPlanarTable.XPlanar_HMI.Status.TileCount
        Textfield (36,84 150x26), "Tile Count"
        Textfield (188,116 69x26), "%d", text variable: MAIN.Machine.XPlanar.XPlanarTable.XPlanar_HMI.Status.NumberOfMovers
        Textfield (36,116 150x26), "Number of Movers"
        Textfield (188,146 69x26), "%d", text variable: MAIN.Machine.XPlanar.XPlanarTable.XPlanar_HMI.Status.NumberOfTracks
        Textfield (36,146 150x26), "Number of Tracks"
        Textfield (188,176 69x26), "%d", text variable: MAIN.Machine.XPlanar.XPlanarTable.XPlanar_HMI.Status.NumberOfStations
        Textfield (36,176 150x26), "Number of Stations"
        GroupBox (0,0 316x220), "XPlanar Table"
END_VISUALIZATION

// ---- StationList_TextList.TcTLO
TEXTLIST StationList_TextList
  0 = 'Process'
  1 = 'Decision'
   = ''
END_TEXTLIST
